# EPICS substitutions: iocBoot/iocEK9KTest/Test3.substitutions
file "../../db/EL2008.template"
{ 	pattern
	{
		TERMINAL,
		DESC1,	ZNAM1,	ONAM1,	PINI1,
		DESC2,	ZNAM2,	ONAM2,	PINI2,
		DESC3,	ZNAM3,	ONAM3,	PINI3,
		DESC4,	ZNAM4,	ONAM4,	PINI4,
		DESC5,	ZNAM5,	ONAM5,	PINI5,
		DESC6,	ZNAM6,	ONAM6,	PINI6,
		DESC7,	ZNAM7,	ONAM7,	PINI7,
		DESC8,	ZNAM8,	ONAM8,	PINI8
	}
	{
		"BO:1",
		"Sig1", "",		"",		"",
		"Sig2", "",		"",		"",
		"Sig3", "",		"",		"",
		"Sig4", "",		"",		"",
		"Sig5", "",		"",		"",
		"Sig6", "",		"",		"",
		"Sig7", "",		"",		"",
		"Sig8", "",		"",		""
	}
}

file "../../db/EL2008.template"
{ 	pattern
	{
		TERMINAL,
		DESC1,	ZNAM1,	ONAM1,	PINI1,
		DESC2,	ZNAM2,	ONAM2,	PINI2,
		DESC3,	ZNAM3,	ONAM3,	PINI3,
		DESC4,	ZNAM4,	ONAM4,	PINI4,
		DESC5,	ZNAM5,	ONAM5,	PINI5,
		DESC6,	ZNAM6,	ONAM6,	PINI6,
		DESC7,	ZNAM7,	ONAM7,	PINI7,
		DESC8,	ZNAM8,	ONAM8,	PINI8
	}
	{
		"BO:2",
		"Sig1", "",		"",		"",
		"Sig2", "",		"",		"",
		"Sig3", "",		"",		"",
		"Sig4", "",		"",		"",
		"Sig5", "",		"",		"",
		"Sig6", "",		"",		"",
		"Sig7", "",		"",		"",
		"Sig8", "",		"",		""
	}
}

file "../../db/EL3054.template"
{ 	pattern
	{
		TERMINAL,
		DESC1,	SCAN1,	ADEL1,	EGUF1,	EGUL1,	HIGH1,	HIHI1,	HOPR1,	HYST1,	LOLO1,	LOPR1,	LOW1,	MDEL1,	SMOO1,	EGU1,
		DESC2,	SCAN2,	ADEL2,	EGUF2,	EGUL2,	HIGH2,	HIHI2,	HOPR2,	HYST2,	LOLO2,	LOPR2,	LOW2,	MDEL2,	SMOO2,	EGU2,
		DESC3,	SCAN3,	ADEL3,	EGUF3,	EGUL3,	HIGH3,	HIHI3,	HOPR3,	HYST3,	LOLO3,	LOPR3,	LOW3,	MDEL3,	SMOO3,	EGU3,
		DESC4,	SCAN4,	ADEL4,	EGUF4,	EGUL4,	HIGH4,	HIHI4,	HOPR4,	HYST4,	LOLO4,	LOPR4,	LOW4,	MDEL4,	SMOO4,	EGU4
	}
	{
		"AI:1",
		"Signal1", ".1 second", "", "20", "4", "",		"",		"",		"",		"",		"",		"",		"",		"",		"mA",
		"Signal2", ".1 second", "", "20", "4", "",		"",		"",		"",		"",		"",		"",		"",		"",		"mA",
		"Signal3", ".1 second", "", "20", "4", "",		"",		"",		"",		"",		"",		"",		"",		"",		"mA",
		"Signal4", ".1 second", "", "20", "4", "",		"",		"",		"",		"",		"",		"",		"",		"",		"mA"
	}
}

file "../../db/EL1004.template"
{ 	pattern
	{
		TERMINAL,
		DESC1,	ZNAM1,	ONAM1,	ZSV1,	OSV1,	COSV1,	SCAN1,
		DESC2,	ZNAM2,	ONAM2,	ZSV2,	OSV2,	COSV2,	SCAN2,
		DESC3,	ZNAM3,	ONAM3,	ZSV3,	OSV3,	COSV3,	SCAN3,
		DESC4,	ZNAM4,	ONAM4,	ZSV4,	OSV4,	COSV4,	SCAN4
	}
	{
		"BI:1",
		"",		"",		"",		"",		"",		"",		".1 second",
		"",		"",		"",		"",		"",		"",		".1 second",
		"",		"",		"",		"",		"",		"",		".1 second",
		"",		"",		"",		"",		"",		"",		".1 second"
	}
}
